(* CODESYS project FU_siBitPartThrough.xml

Project tree, tasks and I/O mapping:
  function FU_siBitPartThrough [ST]
*)

// FU_siBitPartThrough
//This function changed only the needed bits of a variable
// |**Version**|**Author**| **Date** |**Changes**
// | 1         | NSN      | 16-03-22 | Creation
FUNCTION FU_siBitPartThrough : SINT
VAR_INPUT
	valueChange		:SINT;		//Variable to change
	value			:SINT;		//Value to change bits to
	amount			:BYTE;		//Amount of bits to change
	offset			:BYTE;		//Offset in variable to change bits at
END_VAR

FU_siBitPartThrough		:=		TO_SINT((TO_USINT(valueChange) AND ROL(TO_USINT(GConstants.binaryInvMaskSint[amount]),offset)) OR SHL(TO_USINT(value) AND TO_USINT(GConstants.binaryMaskSint[amount]),offset));

END_FUNCTION
